{attribute 'call_after_init'}
FUNCTION_BLOCK FB_SimpleStringBuilder_Test EXTENDS TcUnit.FB_TestSuite IMPLEMENTS TcUnit.I_RunnableTestSuite
VAR
    Assert : TcUnit.FB_Assert;
    
    initializedStringBuilderEmpty_StringBuilder: SimpleStringBuilder;
    
    appendOneString_StringBuilder: SimpleStringBuilder;
    
    appendThreeStrings_StringBuilder: SimpleStringBuilder;
    
    appendINT_StringBuilder: SimpleStringBuilder;
END_VAR

METHOD FB_init : BOOL
VAR_INPUT
	bInitRetains : BOOL; // if TRUE, the retain variables are initialized (warm start / cold start)
	bInCopyCode : BOOL;  // if TRUE, the instance afterwards gets moved into the copy code (online change)
END_VAR
SUPER^.RegisterTestSuite(THIS^);
END_METHOD

METHOD RunTests : TCUNIT.E_TestSuiteRunState
Test_InitializedStringBuilderEmpty();
Test_AppendOneString();
Test_AppendThreeStrings();
Test_AppendINT();

RunTests := TCUNIT.E_TestSuiteRunState.FINISHED;
END_METHOD

METHOD Test_AppendINT
VAR
    expected: STRING(10);
    actual: STRING(10);
    
    testINT: INT;
END_VAR
TEST('Test_AppendINT');

expected := '13';

testINT := 13;
appendINT_StringBuilder.append(testINT);
actual := appendINT_StringBuilder.toString();

Assert.AssertEquals_STRING(expected, actual, 'Appended INT does not match');
END_METHOD

METHOD Test_AppendOneString
VAR
    expected: STRING(10);
    actual: STRING(10);
    
    testString: STRING(10);
END_VAR
TEST('Test_AppendOneString');

expected := 'twincat$R';

testString := 'twincat$R';
appendOneString_StringBuilder.append(testString);
actual := appendOneString_StringBuilder.toString();

Assert.AssertEquals_STRING(expected, actual, 'String did not append');
END_METHOD

METHOD Test_AppendThreeStrings
VAR
    expected: STRING(30);
    actual: STRING(30);
    
    testString1: STRING(10);
    testString2: STRING(10);
    testString3: STRING(10);
END_VAR
TEST('Test_AppendThreeStrings');

expected := 'hello$Tworld$Tfoo$R';

testString1 := 'hello$T';
appendThreeStrings_StringBuilder.append(testString1);
testString2 := 'world$T';
appendThreeStrings_StringBuilder.append(testString2);
testString3 := 'foo$R';
appendThreeStrings_StringBuilder.append(testString3);
actual := appendThreeStrings_StringBuilder.toString();

Assert.AssertEquals_STRING(expected, actual, 'Appended Strings do not match');
END_METHOD

METHOD Test_InitializedStringBuilderEmpty
VAR
    expected: STRING(10);
    actual: STRING(10);
END_VAR
TEST('Test_InitializedStringBuilderEmpty');

expected := '';
actual := initializedStringBuilderEmpty_StringBuilder.toString();

Assert.AssertEquals_STRING(expected, actual, 'Initialized String Builder not empty');
END_METHOD

END_FUNCTION_BLOCK

(* stored: Version 1.1.0.1, ProductVersion 3.1.4022.12
   POU FB_SimpleStringBuilder_Test: Id {2eefe505-04ad-490d-bcce-970863b4c8fe}, SpecialFunc None
   Method FB_init: Id {f8d90e8d-ed56-4ccd-a130-40ffeae34ec8}
   Method RunTests: Id {0babc269-d08a-4fc9-bd35-3df8d318f3fd}
   Method Test_AppendINT: Id {29ca6270-3348-4295-8743-ffdeec11eb68}
   Method Test_AppendOneString: Id {add111b9-c4e0-4aaf-8e6d-44fe73c97f1e}
   Method Test_AppendThreeStrings: Id {2703faa4-71af-44a7-a55a-3e0958b044b3}
   Method Test_InitializedStringBuilderEmpty: Id {c4215bac-3bb1-40f6-8a9c-dd31ee905728} *)
